FUNCTION_BLOCK FB_FileIO
VAR	
	_sNetId				: STRING;
	_sPath				: STRING;
	fbFileOpen 			: FB_FileOpen;
	fbFileWrite 		: FB_FileWrite;
	fbFileRead 			: FB_FileRead;
	fbFileClose 		: FB_FileClose;	
	fbCreateDir			: FB_CreateDir;
	nHFile 				: UINT := 0;
	eReadState 			: E_FileIoState := READY;
	eWriteState 		: E_FileIoState := READY;
	nBytesReadResult	: UDINT;
	nErrorIdResult		: UDINT;	
END_VAR

PROPERTY PUBLIC nBytesRead : UDINT
GET
nBytesRead := nBytesReadResult;
END_GET
SET // PRIVATE
nBytesReadResult := nBytesRead;
END_SET
END_PROPERTY

PROPERTY PUBLIC nErrorId : uDINT
GET
nErrorId := nErrorIdResult;
END_GET
SET // PRIVATE
nErrorIdResult := nErrorId;
END_SET
END_PROPERTY

METHOD PUBLIC Read : BOOL
VAR_INPUT
	sFileName	: T_MaxString;
	pData		: PVOID;
	nLength		: UDINT;
END_VAR
Read := FALSE;
CASE eReadState OF
	E_FileIoState.READY:
		fbFileOpen(sNetId := _sNetId, bExecute := FALSE);
		fbFileRead(sNetId := _sNetId, bExecute := FALSE);
		fbFileClose(sNetId := _sNetId, bExecute := FALSE);
		eReadState := E_FileIoState.OPEN;
		
	E_FileIoState.OPEN:
		nErrorId := 0;
		nBytesRead := 0;
		IF nHFile = 0 THEN
			fbFileOpen.sPathName := sFileName;
			fbFileOpen.nMode := FOPEN_MODEREAD;
			fbFileOpen.ePath := PATH_GENERIC;
			fbFileOpen(bExecute := TRUE);
		END_IF
		IF fbFileOpen.hFile <> 0 AND NOT fbFileOpen.bBusy AND NOT fbFileOpen.bError THEN
			nHFile := fbFileOpen.hFile;
			fbFileOpen(bExecute := FALSE);			
			fbFileRead.hFile := nHFile;
			fbFileRead.cbReadLen := nLength;
			fbFileRead.pReadBuff := pData;
			eReadState := E_FileIoState.READ;
		END_IF
		IF fbFileOpen.bError THEN
			fbFileOpen(bExecute := FALSE);
			nErrorId := fbFileOpen.nErrId;
			eReadState := E_FileIoState.CREATE;
		END_IF
		
	E_FileIoState.CREATE:
		IF THIS^.Write(sFileName, pData, nLength) THEN
			IF nErrorId = 0 THEN
				eReadState := E_FileIoState.OPEN;
			ELSE
				eReadState := E_FileIoState.ERROR;
			END_IF
		END_IF
				
	E_FileIoState.READ:
		fbFileRead(bExecute := TRUE);
		IF NOT fbFileRead.bBusy AND NOT fbFileRead.bError THEN
			nBytesRead := fbFileRead.cbRead;
			fbFileRead(bExecute := FALSE);
			eReadState := E_FileIoState.CLOSE;
		END_IF
		IF fbFileRead.bError THEN
			nErrorId := fbFileRead.nErrId;
			eReadState := E_FileIoState.ERROR;
		END_IF
		
	E_FileIoState.CLOSE:
		IF nHFile <> 0 THEN
			fbFileClose(hFile := nHFile, bExecute := TRUE);
		END_IF
		IF NOT fbFileClose.bBusy THEN
			fbFileClose(bExecute := FALSE);
			nHFile := 0;
			eReadState := E_FileIoState.READY;
			Read := TRUE;
		END_IF
				
	E_FileIoState.ERROR:
		F_LogError(CONCAT('Error reading/writing file in ', CONCAT(_sNetId, CONCAT(' - ', _sPath))));
		eReadState := E_FileIoState.CLOSE;
		
END_CASE
END_METHOD

PROPERTY sNetId : STRING
GET
sNetId := _sNetId;
END_GET
SET
_sNetId := sNetId;
END_SET
END_PROPERTY

PROPERTY sPath : STRING
GET
sPath := _sPath;
END_GET
SET
_sPath := sPath;
END_SET
END_PROPERTY

METHOD PUBLIC Write : BOOL
VAR_INPUT
	sFileName	: T_MaxString;
	pData 		: PVOID;
	nLength 	: UDINT;
END_VAR
Write := FALSE;
CASE eWriteState OF
	E_FileIoState.READY:
		fbFileOpen(sNetId := _sNetId, bExecute := FALSE);
		fbFileWrite(sNetId := _sNetId, bExecute := FALSE);
		fbFileClose(sNetId := _sNetId, bExecute := FALSE);
		fbCreateDir(sNetId := _sNetId, bExecute := FALSE);
		eWriteState := E_FileIoState.OPEN;
		
	E_FileIoState.OPEN:
		nErrorId := 0;
		IF nHFile = 0 THEN
			fbFileOpen.sPathName := sFileName;
			fbFileOpen.nMode := FOPEN_MODEWRITE;
			fbFileOpen.ePath := PATH_GENERIC;
			fbFileOpen(bExecute := TRUE);
		END_IF
		IF fbFileOpen.hFile <> 0 AND NOT fbFileOpen.bBusy AND NOT fbFileOpen.bError THEN
			nHFile := fbFileOpen.hFile;
			fbFileOpen(bExecute := FALSE);					
			fbFileWrite.hFile := nHFile;
			fbFileWrite.cbWriteLen := nLength;
			fbFileWrite.pWriteBuff := pData;
			eWriteState := E_FileIoState.WRITE;
		END_IF
		IF fbFileOpen.bError THEN
			fbFileOpen(bExecute := FALSE);
			nErrorId := fbFileOpen.nErrId;
			eWriteState := E_FileIoState.CREATE;			
		END_IF
		
	E_FileIoState.CREATE:
		fbCreateDir.sPathName:= _sPath;
		fbCreateDir.ePath:= PATH_GENERIC;
		fbCreateDir(bExecute := TRUE);
		IF NOT fbCreateDir.bBusy AND NOT fbCreateDir.bError THEN
			nErrorId := 0;
			fbCreateDir(bExecute := FALSE);
			eWriteState := E_FileIoState.OPEN;
		END_IF
		IF fbCreateDir.bError THEN
			nErrorId := fbCreateDir.nErrId;
			eWriteState := E_FileIoState.ERROR;			
		END_IF
				
	E_FileIoState.WRITE:
		fbFileWrite(bExecute := TRUE);
		IF NOT fbFileWrite.bBusy AND fbFileWrite.cbWrite = nLength AND NOT fbFileWrite.bError THEN
			fbFileWrite(bExecute := FALSE);
			eWriteState := E_FileIoState.CLOSE;
		END_IF
		IF fbFileWrite.bError THEN
			nErrorId := fbFileWrite.nErrId;
			eWriteState := E_FileIoState.ERROR;
		END_IF
		
	E_FileIoState.CLOSE:
		IF  nHFile <> 0 THEN
			fbFileClose(hFile := nHFile, bExecute := TRUE);
		END_IF
		IF NOT fbFileClose.bBusy THEN
			fbFileClose(bExecute := FALSE);
			nHFile := 0;
			eWriteState := E_FileIoState.READY;
			Write := TRUE;
		END_IF

	E_FileIoState.ERROR:
		F_LogError(CONCAT('Error reading/writing file in ', CONCAT(_sNetId, CONCAT(' - ', _sPath))));
		eWriteState := E_FileIoState.CLOSE;	

END_CASE
END_METHOD

END_FUNCTION_BLOCK

(* stored: Version 1.1.0.1, ProductVersion 3.1.4024.12
   POU FB_FileIO: Id {9bd0ee4a-382c-097c-0148-97ed6cb4f83e}, SpecialFunc None
   Property nBytesRead: Id {77d13791-0365-08c4-3bd9-096e691e978b}
   Get Get: Id {f25b037a-82a3-01f6-3927-ed3e9b0a6234}
   Set Set: Id {dd598571-c71e-048c-391c-82a7be85eeae}
   Property nErrorId: Id {cfef08be-643c-0e12-22fb-90630518dad7}
   Get Get: Id {7b8c5cc6-591a-0ab8-1bf5-f9fe8b7ca6c1}
   Set Set: Id {8758247d-9ed6-0698-25af-4a957bc27e4e}
   Method Read: Id {88360398-0c6e-0b7e-0e2d-578c6012dec3}
   Property sNetId: Id {e5323cd2-2532-0a2a-0b62-cd12af0fc498}
   Get Get: Id {b6ab6318-d9d7-062e-0bb5-bd2818d9d253}
   Set Set: Id {3f44aea4-48fe-01ec-2bff-fb9bdaa8d292}
   Property sPath: Id {06934dc8-2694-07cf-16fe-75a309d1c44f}
   Get Get: Id {fbf55ba6-f6f0-0b6f-0ce6-2ff953730a55}
   Set Set: Id {57f28500-383c-07d1-26f1-947f17fbf6b6}
   Method Write: Id {68c59710-200f-05a4-0ce2-66f5a6e5ee04} *)
